FUNCTION F_LogLA6 
VAR_INPUT
	eLogLevel		: E_LogLevel;
	sLogger			: T_MaxString;
	sMessage		: T_MaxString;
	aArg1			: ANY;
	aArg2			: ANY;
	aArg3			: ANY;
	aArg4			: ANY;
	aArg5			: ANY;
	aArg6			: ANY;
END_VAR
VAR 
	aEmptyArg		: BYTE;
END_VAR

F_LogA(
	eLogLevel,
	sLogger,
	sMessage,
	4,
	aArg1,
	aArg2,
	aArg3,
	aArg4,
	aArg5,
	aArg6,
	aEmptyArg,
	aEmptyArg,
	aEmptyArg,
	aEmptyArg
);

END_FUNCTION

(* stored: Version 1.1.0.1, ProductVersion 3.1.4024.0
   POU F_LogLA6: Id {316b3328-3162-4cad-828c-64c859230c23}, SpecialFunc None *)
